TYPE ST_Param :
STRUCT
	stStatus:ST_ParamStatus;//informations d'états (compteur de pièces, modes,...)
	stFixed:ST_ParamFixed;//Paramètres pas en lien avec le produit, fixe
	stRecipe:ST_ParamRecipe;//Paramètres en lien avec le produit
END_STRUCT
END_TYPE

(* stored: Version 1.1.0.1, ProductVersion 3.1.4020.6
   DUT ST_Param: Id {d2cd521b-c212-49e4-9c20-780409e3c8ea} *)
